PROGRAM TSCS_Bridge_Diagnostic
(*Generates a test signal for the bridge terminal then compares it against a readback signal*)
VAR
	TestSignal : REAL;
	
	TDU_TestSignal_Delay :REAL := 0; // Number of counts behind the TDU TestSignal
	TMS_TestSignal_Delay :REAL := 0; // Number of counts behind the TMS TestSignal 
	
	// Parameters
	CountRate : REAL := 1.0; // ms per cycle (e.g. 1.0 for a 1ms excution rate)
	Signal_HL : REAL := 1000; // Signal High Limit
	Signal_LL : REAL := -1000; // Signal Low Limit
 
	RS_0: RS;	// Counter state (Set = Count-DOWN active)
END_VAR
VAR // added by the converter: edge detectors and wires of the graphical bodies
    _rt1, _rt2 : R_TRIG;
END_VAR

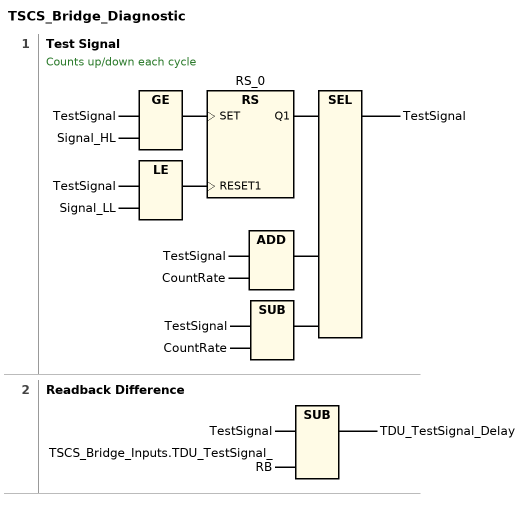
// NETWORK 1: Test Signal
// Counts up/down each cycle
_rt1(CLK := TestSignal >= Signal_HL);
_rt2(CLK := TestSignal <= Signal_LL);
RS_0(SET := _rt1.Q, RESET1 := _rt2.Q); // RS
TestSignal := SEL(RS_0.Q1, TestSignal + CountRate, TestSignal - CountRate);

// NETWORK 2: Readback Difference
TDU_TestSignal_Delay := TestSignal - TSCS_Bridge_Inputs.TDU_TestSignal_RB;

END_PROGRAM

(* stored: Version 1.1.0.1, ProductVersion 3.1.4024.9
   POU TSCS_Bridge_Diagnostic: Id {c2404466-5f35-444f-8eba-adf42f60161e}, SpecialFunc None *)
